FUNCTION_BLOCK FB_HMI
VAR_INPUT
    PLCtoHMI : st_PLCtoHMI;
END_VAR
VAR_OUTPUT
    HMItoPLC : st_HMItoPLC;
END_VAR
VAR
    delayWriteTON : TON := (PT := T#500MS);
    writeDurationTON : TON := (PT := T#50MS);
    //writeJson : BOOL;
END_VAR

IF PLCtoHMI.cell.state = eCellState_Error THEN
    HMItoPLC.hmi.bShowResetBtn := TRUE;
END_IF

IF HMItoPLC.cell.bReset THEN
    HMItoPLC.hmi.bShowResetBtn := FALSE;
END_IF

IF HMItoPLC.cell.bGoToAuto OR HMItoPLC.cell.bGoToManual THEN
    IF PLCtoHMI.cell.state = eCellState_Automatic THEN
        HMItoPLC.cell.bGoToAuto := FALSE;
    END_IF
    IF PLCtoHMI.cell.state = eCellState_Manual THEN
        HMItoPLC.cell.bGoToManual := FALSE;
    END_IF
END_IF

IF PLCtoHMI.variantControl.bNeedsCellDefinition THEN
    IF HMItoPLC.variantControl.bWriteJSON THEN
         delayWriteTON(IN := TRUE);
        IF delayWriteTON.Q THEN
            HMItoPLC.variantControl.bExportJSON := TRUE;
            HMItoPLC.variantControl.bWriteJSON := FALSE;
            delayWriteTON(IN := FALSE);
            writeDurationTON.IN := TRUE;
        END_IF
    END_IF
END_IF

writeDurationTON();
IF writeDurationTON.Q THEN
    HMItoPLC.variantControl.bExportJSON := FALSE;
    writeDurationTON.IN := FALSE;
END_IF

END_FUNCTION_BLOCK

(* stored: Version 1.1.0.1, ProductVersion 3.1.4024.9
   POU FB_HMI: Id {d4e0be77-d28b-42bb-b1c3-1050a081e7a4}, SpecialFunc None *)
